# EPICS substitutions: softIntApp/Db/softInt-asta.substitutions
file highOnFault.template {
pattern
{ N,              INP, LOLIM, HILIM,              OUT}
{01, "ESB:GP01:VAL01",  1e-3,   1e3, "ESB:GP01:VAL02"}
}
